// AUTO mode chain (Core §6.2/§6.8 ST skeleton on FB_SequenceBase): the continuous
// production cycle — await a fresh two-hand start with part+air present, transfer
// the part in, press for the recipe dwell, return to load position, count the good
// part, and loop until Stop. A Stop requested at the between-cycles wait is honored
// there (M_StopNow) so no phantom cycle is charged. Every child motion goes through
// the §6.1 handshake (M_TryIssue); progression rides the shared _retVal.
FUNCTION_BLOCK FB_PressDemoAuto EXTENDS FB_SequenceBase
VAR
    _partReady, _airReady, _startReady : BOOL;
    _dwellTwoHandHeld : BOOL;          // N220 named wait: two-hand held through the dwell
    _decisionRequest : ST_DecisionRequest;   // §6.11 not-reached confirmation
    _answer : INT;
    _ramReached, _failureConfirmed : BOOL;   // N200/N210 named waits
    _twoHandHeldDuringClose : BOOL;          // N180 named wait
    _closeAbortWarned : BOOL;                // N180 §6.9(e) message result
    _ramFailureReported : BOOL;              // N200 §6.9(e) message result
    _partInMachine : BOOL;                   // §3.16.3 the part is already received
    _partDispositioned : BOOL;               // N260 already set the verdict
    _traceAccepted, _recordAccepted, _partProcessed : BOOL;
    {attribute 'OPC.UA.DA' := '0'}
    _pressRam : REFERENCE TO FB_CylinderCM;
    {attribute 'OPC.UA.DA' := '0'}
    _door : REFERENCE TO FB_CylinderCM;
    {attribute 'OPC.UA.DA' := '0'}
    _partSlide : REFERENCE TO FB_CylinderCM;
    {attribute 'OPC.UA.DA' := '0'}
    _twoHand : REFERENCE TO FB_TwoHandStartCM;
    {attribute 'OPC.UA.DA' := '0'}
    _partPresentSensor : REFERENCE TO FB_DigitalInputCM;
    {attribute 'OPC.UA.DA' := '0'}
    _airPressureMonitor : REFERENCE TO FB_AirPressureMonitorCM;
    {attribute 'OPC.UA.DA' := '0'}
    _parCfg : REFERENCE TO ST_PneumaticPressParCfg;
    // §3.8a - the CELL's own policy, held separately from the MODEL's data and
    // referenced exactly like _parCfg, so each step reads whichever structure
    // actually owns the value it is asking about.
    {attribute 'OPC.UA.DA' := '0'}
    _stationCfg : REFERENCE TO ST_PneumaticPressStationCfg;
    {attribute 'OPC.UA.DA' := '0'}
    _outCmd : REFERENCE TO ST_PneumaticPressOutCmd;
    {attribute 'OPC.UA.DA' := '0'}
    _startLatched : REFERENCE TO BOOL;
    {attribute 'OPC.UA.DA' := '0'}
    _loadPosition : FB_PressDemoLoadPosition;
END_VAR

// §6.8 - the chain's own state on a restart (the base resets the flow state).
METHOD PROTECTED OnChainReset
// A chart restart abandons whatever the cycle was holding: the part record is
// closed by N215/N999, never by a restart, so both trackers start clean.
_partDispositioned := FALSE;
_partInMachine := FALSE;
END_METHOD

METHOD M_Run
IF NOT _attached THEN
    RETURN;
END_IF
CASE _step OF
    0:  // initialize
        M_Step(StepNo := 0, StepName := 'project.step.pressAutoInitialize',
            Awaits := 0, AwaitingLabel := '', TimeClass := E_TimeClass.WORK, ExpectedTime := T#0S, Branch := 0);
        _outCmd.CycleCompleted := FALSE;
        _retVal := E_StepResult.ADVANCE;
        M_Advance(OnAdvance := 100, OnJump1 := -1, OnJump2 := -1, OnJump3 := -1 );
    100:  // await a fresh two-hand start (the §8.11.1 cycle-start marker)
        M_Step(StepNo := 100, StepName := 'project.step.pressAwaitTwoHand',
            Awaits := 0, AwaitingLabel := '', TimeClass := E_TimeClass.WAIT_OPERATOR, ExpectedTime := T#0S, Branch := 0);
        _outCmd.CycleCompleted := FALSE;
        _partReady := M_Await(Idx := 1, Label := 'project.condition.partPresent',
            Ok := _partPresentSensor.OutImm.Value AND _partPresentSensor.OutImm.Quality);
        _airReady := M_Await(Idx := 2, Label := 'project.condition.airPressureOk',
            Ok := _airPressureMonitor.OutImm.PressureOk);
        IF _stationCfg.RequireTwoHandStart THEN
            _startReady := M_Await(Idx := 3, Label := 'project.condition.twoHandStart', Ok := _startLatched);
        ELSE
            _startReady := TRUE;
        END_IF
        IF M_StopPending() THEN
            M_StopNow();                       // stop accepted BETWEEN cycles: no phantom cycle
        ELSIF _partReady AND _airReady AND _startReady THEN
            // §3.16.3 receive once per PHYSICAL part. The N180 two-hand abort returns
            // here with the same part still in the machine and nothing processed, so a
            // second M_PartReceived would open a duplicate record for one part.
            // M_PartStarted (N150) is deliberately NOT guarded: each pass is a genuine
            // processing attempt on that part.
            IF NOT _partInMachine THEN
                _traceAccepted := M_PartReceived();
                _partInMachine := TRUE;
            END_IF
            _retVal := E_StepResult.ADVANCE;
        END_IF
        M_Advance(OnAdvance := 110, OnJump1 := -1, OnJump2 := -1, OnJump3 := -1);
    110:  // ram up
        M_Step(StepNo := 110, StepName := 'project.step.pressRamUp',
            Awaits := _pressRam, AwaitingLabel := 'PressRam.RETRACT', TimeClass := E_TimeClass.WORK, ExpectedTime := T#0S, Branch := 0);
        IF M_TryIssue(Steppable := TRUE) THEN
            _pressRam.Abort := FALSE; _pressRam.Command := E_CylinderCommand.RETRACT; _pressRam.Execute := TRUE;
        END_IF
        IF _pressRam.Done THEN _pressRam.Execute := FALSE; _retVal := E_StepResult.ADVANCE; END_IF
        M_Advance(OnAdvance := 130, OnJump1 := -1, OnJump2 := -1, OnJump3 := -1);
    130:  // door open
        M_Step(StepNo := 130, StepName := 'project.step.pressDoorOpen',
            Awaits := _door, AwaitingLabel := 'Door.RETRACT', TimeClass := E_TimeClass.WORK, ExpectedTime := T#0S, Branch := 0);
        IF M_TryIssue(Steppable := TRUE) THEN
            _door.Abort := FALSE; _door.Command := E_CylinderCommand.RETRACT; _door.Execute := TRUE;
        END_IF
        IF _door.Done THEN _door.Execute := FALSE; _retVal := E_StepResult.ADVANCE; END_IF
        M_Advance(OnAdvance := 150, OnJump1 := -1, OnJump2 := -1, OnJump3 := -1);
    150:  // slide inside (value-adding sequence begins)
        M_Step(StepNo := 150, StepName := 'project.step.pressSlideInside',
            Awaits := _partSlide, AwaitingLabel := 'PartSlide.EXTEND', TimeClass := E_TimeClass.WORK, ExpectedTime := T#0S, Branch := 0);
        IF M_TryIssue(Steppable := TRUE) THEN
            M_PartStarted();
            _partSlide.Abort := FALSE; _partSlide.Command := E_CylinderCommand.EXTEND; _partSlide.Execute := TRUE;
        END_IF
        IF _partSlide.Done THEN _partSlide.Execute := FALSE; _retVal := E_StepResult.ADVANCE; END_IF
        M_Advance(OnAdvance := 170, OnJump1 := -1, OnJump2 := -1, OnJump3 := -1);
    170:  // transfer settle
        M_Step(StepNo := 170, StepName := 'project.step.pressTransferSettle',
            Awaits := 0, AwaitingLabel := '', TimeClass := E_TimeClass.WORK, ExpectedTime := _parCfg.TransferSettleTime, Branch := 0);
        _retVal := M_Delay(PT := _parCfg.TransferSettleTime);
        M_Advance(OnAdvance := 180, OnJump1 := -1, OnJump2 := -1, OnJump3 := -1);
    180:  // door close. Releasing a two-hand button while the door is moving is an
          // operator abort, not a fault: the door goes back up, the part slides out,
          // and the cycle returns to the two-hand wait (§6.10 jump). Completion wins
          // if the door finished in the same scan the button was released.
        M_Step(StepNo := 180, StepName := 'project.step.pressDoorClose',
            Awaits := _door, AwaitingLabel := 'Door.EXTEND', TimeClass := E_TimeClass.WORK, ExpectedTime := T#0S, Branch := 0);
        _twoHandHeldDuringClose := M_Await(Idx := 1,
            Label := 'project.condition.twoHandHeldDuringDoorClose',
            Ok := _twoHand.OutImm.SafeActive OR NOT _stationCfg.RequireTwoHandStart);
        IF M_TryIssue(Steppable := TRUE) THEN
            _door.Abort := FALSE; _door.Command := E_CylinderCommand.EXTEND; _door.Execute := TRUE;
        END_IF
        IF _door.Done THEN
            _door.Execute := FALSE;
            _retVal := E_StepResult.ADVANCE;
        ELSIF NOT _twoHandHeldDuringClose THEN
            _door.Execute := FALSE;             // §6.1 Execute-drop reset releases the close
            // §6.9(e) — a WARNING, not a fault: the release is designed operator
            // behaviour and the chain already owns the recovery below, so nothing
            // stops. It is recorded because a cycle was abandoned with the part
            // still in the machine, and the §3.13 chart marks this step for it.
            // The base raises it once per visit however many scans this runs.
            _closeAbortWarned := M_RaiseWarning(
                Reason := PL_PressReasons.PRESS_TWO_HAND_RELEASED,
                DescriptionKey := 'project.warning.twoHandReleasedDuringDoorClose',
                Severity := E_Severity.LOW, Category := E_Category.PROCESS);
            _retVal := E_StepResult.JUMP1;      // released -> reopen and clear the part
        END_IF
        M_Advance(OnAdvance := 200, OnJump1 := 185, OnJump2 := -1, OnJump3 := -1);
    185:  // two-hand released during closing: take the door back up
        M_Step(StepNo := 185, StepName := 'project.step.pressDoorReopen',
            Awaits := _door, AwaitingLabel := 'Door.RETRACT', TimeClass := E_TimeClass.WORK, ExpectedTime := T#0S, Branch := 0);
        IF M_TryIssue(Steppable := TRUE) THEN
            _door.Abort := FALSE; _door.Command := E_CylinderCommand.RETRACT; _door.Execute := TRUE;
        END_IF
        IF _door.Done THEN _door.Execute := FALSE; _retVal := E_StepResult.ADVANCE; END_IF
        M_Advance(OnAdvance := 190, OnJump1 := -1, OnJump2 := -1, OnJump3 := -1);
    190:  // slide the part back out, then return to the two-hand wait. The start latch
          // is dropped so the cycle cannot resume without a fresh two-hand press.
        M_Step(StepNo := 190, StepName := 'project.step.pressSlideOutsideAfterAbort',
            Awaits := _partSlide, AwaitingLabel := 'PartSlide.RETRACT', TimeClass := E_TimeClass.WORK, ExpectedTime := T#0S, Branch := 0);
        IF M_TryIssue(Steppable := TRUE) THEN
            _partSlide.Abort := FALSE; _partSlide.Command := E_CylinderCommand.RETRACT; _partSlide.Execute := TRUE;
        END_IF
        IF _partSlide.Done THEN
            _partSlide.Execute := FALSE;
            _startLatched := FALSE;
            _retVal := E_StepResult.ADVANCE;
        END_IF
        M_Advance(OnAdvance := 100, OnJump1 := -1, OnJump2 := -1, OnJump3 := -1);
    200:  // ram down. THIS step owns the not-reached disposition, so it does NOT hand
          // the ram to the §6.9 auto-rollup: an awaited child fault is adopted by the
          // Unit (ERROR, _step := 0) before _M_Dispatch runs, and the chain would stop
          // before it could ask the operator anything. The wait is still named (§6.9(b))
          // and the cylinder still raises its own CYL_NOT_EXTENDED alarm.
        M_Step(StepNo := 200, StepName := 'project.step.pressRamDown',
            Awaits := 0, AwaitingLabel := '', TimeClass := E_TimeClass.WORK, ExpectedTime := T#0S, Branch := 0);
        _ramReached := M_Await(Idx := 1, Label := 'project.condition.pressRamExtended',
            Ok := _pressRam.Done);
        IF M_TryIssue(Steppable := TRUE) THEN
            _pressRam.Abort := FALSE; _pressRam.Command := E_CylinderCommand.EXTEND; _pressRam.Execute := TRUE;
        END_IF
        IF _pressRam.Done THEN
            _pressRam.Execute := FALSE;
            _retVal := E_StepResult.ADVANCE;
        ELSIF _pressRam.Error THEN
            // §6.9(e) — publish the ram's own first-out (CYL_NOT_EXTENDED, with its
            // text and IO tag) on the Unit and on this row of the §3.13 chart, and
            // do NOT adopt it: the confirmation + scrap below IS the handling, so a
            // fault here would replace a designed recovery. Saying nothing is what
            // left the failure visible only on the ram itself.
            _ramFailureReported := M_ReportFromChild(Source := _pressRam);
            _pressRam.Execute := FALSE;         // §6.1 Execute-drop reset returns the ram to READY
            _retVal := E_StepResult.JUMP1;      // did not reach -> operator confirmation
        END_IF
        M_Advance(OnAdvance := 220, OnJump1 := 210, OnJump2 := -1, OnJump3 := -1);
    210:  // press did not reach: the operator confirms the failure before the part is
          // scrapped. A scrap is deliberate, so there is no timeout default (§6.11).
        M_Step(StepNo := 210, StepName := 'project.step.pressNotReachedConfirm',
            Awaits := 0, AwaitingLabel := '', TimeClass := E_TimeClass.WAIT_OPERATOR, ExpectedTime := T#0S, Branch := 0);
        _decisionRequest.Prompt := 'project.decision.pressNotReached';
        _decisionRequest.Options[1] := 'project.decision.confirmScrapAndReturn';
        _decisionRequest.Default := 0;
        _decisionRequest.Timeout := T#0S;
        M_AskDecision(Req := _decisionRequest);
        _answer := M_TakeDecision();
        IF _answer = 1 THEN
            _retVal := E_StepResult.ADVANCE;
        ELSE
            _failureConfirmed := M_Await(Idx := 1,
                Label := 'project.condition.pressFailureConfirmation', Ok := FALSE);
        END_IF
        M_Advance(OnAdvance := 215, OnJump1 := -1, OnJump2 := -1, OnJump3 := -1);
    215:  // disposition the part NOK, then rejoin the shared return-to-start step
        M_Step(StepNo := 215, StepName := 'project.step.pressScrapPart',
            Awaits := 0, AwaitingLabel := '', TimeClass := E_TimeClass.WORK, ExpectedTime := T#0S, Branch := 0);
        _partProcessed := M_PartProcessed(Verdict := E_Verdict.NOK,
            Reason := PL_ModuleReasons.CYL_NOT_EXTENDED);
        _partDispositioned := TRUE;             // N999 must not also count it good
        _partInMachine := FALSE;                // dispositioned: the next one is a new part
        _outCmd.CycleCompleted := FALSE;
        _retVal := E_StepResult.ADVANCE;
        M_Advance(OnAdvance := 240, OnJump1 := -1, OnJump2 := -1, OnJump3 := -1);
    220:  // press dwell — two-hand must stay held; releasing it HOLDS the dwell
        M_Step(StepNo := 220, StepName := 'project.step.pressDwell',
            Awaits := 0, AwaitingLabel := '', TimeClass := E_TimeClass.WORK, ExpectedTime := _parCfg.PressSettleTime, Branch := 0);
        // Releasing the button mid-dwell is the designed way to stop pressing, so it
        // is a named wait (§6.9(b)), not a fault: the ram's outputs come off, the
        // dwell timer freezes where it is because M_Delay is not called, and pressing
        // again restores the force and finishes the remaining dwell. Faulting here
        // charged an unrecoverable downtime event for normal operator behaviour.
        _dwellTwoHandHeld := M_Await(Idx := 1, Label := 'project.condition.twoHandHeldDuringPress',
            Ok := _twoHand.OutImm.SafeActive OR NOT _stationCfg.RequireTwoHandStart);
        IF NOT _dwellTwoHandHeld THEN
            _pressRam.WithdrawOutputs();
        ELSE
            // The press force is the valve latched by the EXTEND that step 200 already
            // completed, so after a withdraw only this call re-energizes it — and the
            // ram re-checks its own extend permit before it does (§7.2).
            _pressRam.RestoreOutputs();
            _retVal := M_Delay(PT := _parCfg.PressSettleTime);
        END_IF
        M_Advance(OnAdvance := 230, OnJump1 := -1, OnJump2 := -1, OnJump3 := -1);
    230:  // record the applied dwell (§3.16.1 measured value)
        M_Step(StepNo := 230, StepName := 'project.step.pressRecordResult',
            Awaits := 0, AwaitingLabel := '', TimeClass := E_TimeClass.WORK, ExpectedTime := T#0S, Branch := 0);
        _recordAccepted := M_PartRecord(RecordName := 'PressDwell',
            Value := DINT_TO_LREAL(TIME_TO_DINT(_parCfg.PressSettleTime)),
            Minimum := 0, Maximum := 30000,
            Target := DINT_TO_LREAL(TIME_TO_DINT(_parCfg.PressSettleTime)), EngUnit := 'ms');
        _retVal := E_StepResult.ADVANCE;
        M_Advance(OnAdvance := 240, OnJump1 := -1, OnJump2 := -1, OnJump3 := -1);
    240:  // return to the shared load-safe position (composite step)
        _retVal := M_RunSub(Chain := _loadPosition, BaseStepNo := 240);
        M_Advance(OnAdvance := 999, OnJump1 := -1, OnJump2 := -1, OnJump3 := -1);
    999:  // cycle complete — write result, count by verdict, loop (§8.11.1 finish marker)
        M_Step(StepNo := 999, StepName := 'project.step.pressAutoComplete',
            Awaits := 0, AwaitingLabel := '', TimeClass := E_TimeClass.WORK, ExpectedTime := T#0S, Branch := 0);
        _outCmd.CycleCompleted := TRUE;
        IF _partDispositioned THEN
            _partDispositioned := FALSE;       // N260 already set the NOK verdict
        ELSE
            _partProcessed := M_PartProcessed(Verdict := E_Verdict.OK, Reason := E_Reason.NONE);
            IF NOT _partProcessed THEN
                M_CountGood();                 // §3.9: no carrier configured — count directly
            END_IF
        END_IF
        _partInMachine := FALSE;               // processed: the next one is a new part
        _startLatched := FALSE;
        IF M_EndOfCycle() THEN
            _retVal := E_StepResult.ADVANCE;   // stop NOT requested: loop to N100
        END_IF
        M_Advance(OnAdvance := 100, OnJump1 := -1, OnJump2 := -1, OnJump3 := -1);
ELSE
    M_Fault(Reason := E_Reason.STEP_STALLED, DescriptionKey := 'std.error.undefinedStep');
END_CASE
END_METHOD

METHOD Setup : BOOL
VAR_INPUT
    Host : I_SequenceHost;
END_VAR
VAR_IN_OUT
    PressRam : FB_CylinderCM;
    Door : FB_CylinderCM;
    PartSlide : FB_CylinderCM;
    TwoHand : FB_TwoHandStartCM;
    PartPresentSensor : FB_DigitalInputCM;
    AirPressureMonitor : FB_AirPressureMonitorCM;
    ParCfg : ST_PneumaticPressParCfg;
    StationCfg : ST_PneumaticPressStationCfg;
    OutCmd : ST_PneumaticPressOutCmd;
    StartLatched : BOOL;
END_VAR
_pressRam REF= PressRam;
_door REF= Door;
_partSlide REF= PartSlide;
_twoHand REF= TwoHand;
_partPresentSensor REF= PartPresentSensor;
_airPressureMonitor REF= AirPressureMonitor;
_parCfg REF= ParCfg;
_stationCfg REF= StationCfg;
_outCmd REF= OutCmd;
_startLatched REF= StartLatched;
Setup := M_Attach(Host := Host) AND __ISVALIDREF(_pressRam) AND __ISVALIDREF(_door)
    AND __ISVALIDREF(_partSlide) AND __ISVALIDREF(_twoHand)
    AND __ISVALIDREF(_partPresentSensor) AND __ISVALIDREF(_airPressureMonitor)
    AND __ISVALIDREF(_parCfg) AND __ISVALIDREF(_outCmd) AND __ISVALIDREF(_startLatched)
    AND _loadPosition.Setup(Host := Host, PressRam := PressRam, Door := Door, PartSlide := PartSlide);
END_METHOD

END_FUNCTION_BLOCK

(* stored: Version 1.1.0.1, ProductVersion 3.1.4024.16
   POU FB_PressDemoAuto: Id {27be7602-c702-dcca-822f-fb9fc2c74001}, SpecialFunc None
   Method OnChainReset: Id {27be7602-c702-dcca-822f-fb9fc2c74003}
   Method M_Run: Id {27be7602-c702-dcca-822f-fb9fc2c74004}
   Method Setup: Id {27be7602-c702-dcca-822f-fb9fc2c74002} *)
